VAR_GLOBAL // OUTPUTS
    out_hw_lamp_bit AT %Q16.6: BOOL;
END_VAR

(* stored: ProductVersion 3.1.0.18, Version 1.1.0.1 *)
